{attribute addProperty BoxType "EL6201-0000-0017"}
{attribute addProperty Id "Slave_3A_DO0BIT10.12517Slave_3A_DO1BIT10.12518Slave_3A_DO2BIT10.12519Slave_3A_DO3BIT10.12520Slave_3B_DO0BIT10.12521Slave_3B_DO1BIT10.12522Slave_3B_DO2BIT10.12523Slave_3B_DO3BIT10.12524"}
{attribute addProperty CRC "1613846079"}
{attribute addProperty SizeInBites "8"}
{attribute addProperty SizeInBytes "1"}
TYPE Slave_3_Outputs_6031563F :
STRUCT
	{attribute addProperty Name "Slave_3A_DO0"}
	Slave_3A_DO0 : BIT;
	{attribute addProperty Name "Slave_3A_DO1"}
	Slave_3A_DO1 : BIT;
	{attribute addProperty Name "Slave_3A_DO2"}
	Slave_3A_DO2 : BIT;
	{attribute addProperty Name "Slave_3A_DO3"}
	Slave_3A_DO3 : BIT;
	{attribute addProperty Name "Slave_3B_DO0"}
	Slave_3B_DO0 : BIT;
	{attribute addProperty Name "Slave_3B_DO1"}
	Slave_3B_DO1 : BIT;
	{attribute addProperty Name "Slave_3B_DO2"}
	Slave_3B_DO2 : BIT;
	{attribute addProperty Name "Slave_3B_DO3"}
	Slave_3B_DO3 : BIT;
END_STRUCT
END_TYPE

(* stored: Version 1.2.0.0, ProductVersion 3.1.4024.9
   DUT Slave_3_Outputs_6031563F: Id {c85d0855-184a-425a-a726-16daa2c1aed3} *)
